{attribute 'qualified_only'}
VAR_GLOBAL CONSTANT	
		//control mode number for UI
		g_controlModeNum:INT:=9;
		
		//DH joint angle at initial position
		g_jntDHInitPos:ARRAY[1..2,1..7] OF LREAL:=[0,-pi/2,pi/2,-pi,pi,-pi/2,0,      0,-pi/2,pi/2,0,pi,pi/2,0];
		
		//Test points for the spatial cube, with specific locations given by MATLAB
        g_testPointNum:INT:=8;	
		
		//test motion cycle number
		g_testMotCycNum:INT:=20;
		
		//global variables
		g_mArmNum :INT := 2;	
		g_mJntNum:INT:=7;		
		g_deg2Rad :LREAL := pi/180.0;
		
		//DH joint minmum position
		g_minJntDHPos:ARRAY[1..2,1..7] OF LREAL:=[-60*g_deg2Rad, -60*g_deg2Rad-pi/2,  -45*g_deg2Rad+pi/2, -150*g_deg2Rad-pi,  -135*g_deg2Rad+pi,  -62*g_deg2Rad-pi/2, -150*g_deg2Rad,
																						-60*g_deg2Rad, -60*g_deg2Rad-pi/2,  -45*g_deg2Rad+pi/2,  -90*g_deg2Rad,    -135*g_deg2Rad+pi,    -242*g_deg2Rad+pi/2, -150*g_deg2Rad];
		
		//DH joint minmum position
		g_maxJntDHPos:ARRAY[1..2,1..7] OF LREAL:=[60*g_deg2Rad,	 60*g_deg2Rad-pi/2,   40*g_deg2Rad+pi/2,  90*g_deg2Rad-pi,    135*g_deg2Rad+pi,  242*g_deg2Rad-pi/2, 150*g_deg2Rad,
																						60*g_deg2Rad,	 60*g_deg2Rad-pi/2,   40*g_deg2Rad+pi/2,   150*g_deg2Rad,    135*g_deg2Rad+pi,     62*g_deg2Rad+pi/2, 150*g_deg2Rad];
																			
		//data number for record and write													
		g_recordDataNum:INT:=13000;
		g_writeDataNum:INT:=5500;
		
		
		
		
		//Accuracy testing points under the condition of unchanged posture
		//Test sequence:C-D-H-G-B-A-E-F
		//If testing the accuracy of a single arm, it is necessary to test point by point
		//If testing master-slave accuracy, it is necessary to test point by point
		g_armPoseA1:ARRAY [1..8,1..7] OF LREAL:=[
			0.1341,   -0.2232,    0.1479,   1.5708,0,-1.5708,0,
			0.3136,   -0.3808,    0.1698,   1.5708,0,-1.5708,0,
			0.3136,   -0.3808,    0.5270,   1.5708,0,-1.5708,0,
			0.1341,   -0.2232,    0.540,   1.5708,0,-1.5708,0,
			0.2498,    0.0735,     0.0626,   1.5708,0,-1.5708,0,
			0.4060,    0.0735,     0.0474,   1.5708,0,-1.5708,0,
			0.4060,    0.0735,     0.5716,   1.5708,0,-1.5708,0,
			0.2498,    0.0735,     0.530,   1.5708,0,-1.5708,0];
		g_armPoseA2:ARRAY [1..8,1..7] OF LREAL:=[
			0.2498,    -0.0735,     0.0626,   1.5708,0,-1.5708,0,
			0.4060,    -0.0735,     0.0474,   1.5708,0,-1.5708,0,
			0.4060,    -0.0735,     0.5716,   1.5708,0,-1.5708,0,
			0.2498,    -0.0735,     0.5196,   1.5708,0,-1.5708,0,
			0.1341,     0.2232,     0.1479,   1.5708,0,-1.5708,0,
			0.3136,      0.3808,     0.1698,   1.5708,0,-1.5708,0,
			0.3136,      0.3808,     0.4870,   1.5708,0,-1.5708,0,
			0.1341,      0.2232,     0.4720,   1.5708,0,-1.5708,0];			
	
	
	(*
		//Maximum workspace testing related points
		g_maxSpaceArm1:ARRAY [1..8,1..7] OF LREAL:=[
			0.41371,   0.0785,  0.0454,   1.5708,    0.0000,   -1.5708,0,
			0.24851,   0.0785, 0.06149,   1.5708,   -0.1745,   -1.5708,0,
			0.13024, -0.22483,  0.1403,   1.5680,    0.1775,   -1.5714,0,
			0.31312, -0.38287, 0.15757,   1.5708,    0.0000,   -1.3963,0,
			0.41371,   0.0785, 0.57824,  1.5708,   -0.0000,   -1.7453,0,
			0.24851,   0.0785, 0.52214,  1.7453,   -0.0000,   -1.5708,0,
			0.13089, -0.22316, 0.47087,  1.3963,    0.0000,   -1.5708,0,
			0.31358, -0.38078, 0.52699,  1.5708,   -0.0873,   -1.5708,0];
		g_maxSpaceArm2:ARRAY [1..8,1..7] OF LREAL:=[
			0.41371, -0.0785,  0.0454,   1.5708,    0.0000,   -1.5708,0,
			0.24851, -0.0785, 0.06149,   1.5708,   -0.1745,   -1.5708,0,
			0.13024, 0.22483,  0.1403,   1.5708,    0.1745,   -1.5708,0,
			0.31312, 0.38287, 0.15757,   1.5708,   -0.0000,   -1.3963,0,
			0.41371, -0.0785, 0.57824,   1.5708,    0.0000,   -1.7453,0,
			0.24851, -0.0785, 0.52214,  1.3963,   -0.0000,   -1.5708,0,
			0.13089, 0.22316, 0.47087,  1.6698,    -0.086,   -1.5792,0,
			0.31358, 0.38078, 0.52699,  1.5708,   -0.0873,   -1.5708,0];		
	*)
	

		//testing points for ESD test
		g_esdPoseA1:ARRAY [1..8,1..7] OF LREAL:=[
			0.2333,   -0.1469,    0.2715,   1.5708,0,-1.5708,0,
			0.2872,   -0.1942,    0.2781,   1.5708,0,-1.5708,0,
			0.2872,   -0.1942,    0.3853,   1.5708,0,-1.5708,0,
			0.2333,   -0.1469,    0.3892,   1.5708,0,-1.5708,0,
			0.2681,   -0.0579,    0.2460,   1.5708,0,-1.5708,0,
			0.3149,   -0.0579,    0.2414,   1.5708,0,-1.5708,0,
			0.3149,   -0.0579,    0.3987,   1.5708,0,-1.5708,0,
			0.2681,   -0.0579,    0.3862,   1.5708,0,-1.5708,0];
		g_esdPoseA2:ARRAY [1..8,1..7] OF LREAL:=[
			0.2681,    0.0579,    0.2356,   1.5708,0,-1.5708,0,
			0.3149,    0.0579,    0.2310,   1.5708,0,-1.5708,0,
			0.3149,    0.0579,    0.3883,   1.5708,0,-1.5708,0,
			0.2681,    0.0579,    0.3727,   1.5708,0,-1.5708,0,
			0.2333,    0.1469,    0.2612,   1.5708,0,-1.5708,0,
			0.2872,    0.1942,    0.2678,   1.5708,0,-1.5708,0,
			0.2872,    0.1942,    0.3629,   1.5708,0,-1.5708,0,
			0.2333,    0.1469,    0.3584,   1.5708,0,-1.5708,0];	
			
			
			
		//******************************test data*******************************//
		//Maximum workspace testing related points
		g_maxSpaceArm1:ARRAY [1..8,1..7] OF LREAL:=[
			0.41371,   0.0785,  0.0424,   1.5708,    0.0000,   -1.5708,0,
			0.246,   0.0785,   0.059,   1.5708,   -0.1745,   -1.5708,0,
			0.13024, -0.22483,  0.1403,   1.5680,    0.1775,   -1.5714,0,
			0.318, -0.38287, 0.15757,   1.5708,    0.0000,   -1.3963,0,
			0.41371,   0.0785, 0.57824,  1.5708,   -0.0000,   -1.7453,0,
			0.246,   0.0785, 0.52214,  1.7453,   -0.0000,   -1.5708,0,
			0.13, -0.22316,   0.473,  1.3963,    0.0000,   -1.5708,0,
			0.315,   -0.382, 0.52699,  1.5708,   -0.0873,   -1.5708,0];
		g_maxSpaceArm2:ARRAY [1..8,1..7] OF LREAL:=[
			0.41371, -0.0785,  0.0424,   1.5708,    0.0000,   -1.5708,0,
			0.246, -0.0785,   0.059,   1.5708,   -0.1745,   -1.5708,0,
			0.13024, 0.22483,  0.1403,   1.5708,    0.1745,   -1.5708,0,
			0.318, 0.38287, 0.15757,   1.5708,   -0.0000,   -1.3963,0,
			0.41371, -0.0785, 0.57824,   1.5708,    0.0000,   -1.7453,0,
			0.246, -0.0785, 0.52214,  1.3963,   -0.0000,   -1.5708,0,
			0.13, 0.22316,   0.473,  1.6698,    -0.086,   -1.5792,0,
			0.315,   0.382, 0.52699,  1.5708,   -0.0873,   -1.5708,0];			
END_VAR

(* stored: Version 1.1.0.1, ProductVersion 3.1.4024.11
   GVL GVL_Const: Id {cf747bed-c98f-4034-9edf-cccd140613d8} *)
